FUNCTION_BLOCK StatusLight (* Composite Function Block Type *)
  (* Standard: 61499-2 *)
  (* Version 0.0, 2015-05-20, 4DIAC-IDE, 4DIAC-Consortium *)
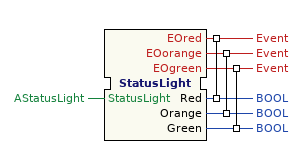
  EVENT_OUTPUT
    EOred WITH Red; (* Execution Confirmation *)
    EOorange WITH Orange;
    EOgreen WITH Green;
  END_EVENT
  VAR_OUTPUT
    Red : BOOL; (* Output event qualifier *)
    Orange : BOOL;
    Green : BOOL;
  END_VAR
  SOCKETS
    StatusLight : AStatusLight;
  END_SOCKETS
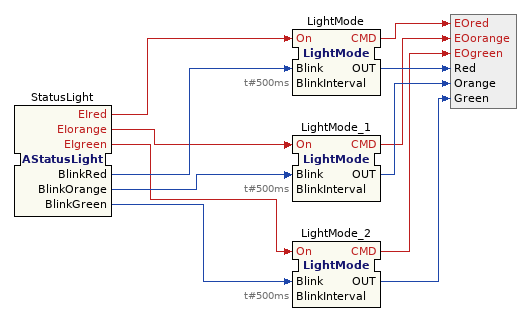
  FBS
    LightMode : LightMode(BlinkInterval := t#500ms);
    LightMode_1 : LightMode(BlinkInterval := t#500ms);
    LightMode_2 : LightMode(BlinkInterval := t#500ms);
  END_FBS
  EVENT_CONNECTIONS
    LightMode.CMD TO EOred;
    LightMode_1.CMD TO EOorange;
    LightMode_2.CMD TO EOgreen;
    StatusLight.EIred TO LightMode.On;
    StatusLight.EIorange TO LightMode_1.On;
    StatusLight.EIgreen TO LightMode_2.On;
  END_CONNECTIONS
  DATA_CONNECTIONS
    LightMode.OUT TO Red;
    LightMode_1.OUT TO Orange;
    LightMode_2.OUT TO Green;
    StatusLight.BlinkRed TO LightMode.Blink;
    StatusLight.BlinkOrange TO LightMode_1.Blink;
    StatusLight.BlinkGreen TO LightMode_2.Blink;
  END_CONNECTIONS
END_FUNCTION_BLOCK
